FUNCTION_BLOCK EQ_Plunger (* Linear actuator through an L298N (IN1 retract, IN2 extend); no sensors. ENA (200/255 on the ESP32) is tied to 3.3 V on the Pi, which has only two hardware PWM channels, so it runs at full speed; equipment IO: owns its IO points; commands Stop=0, Extend=1, Retract=2 *)
  (* Standard: 61499-2 *)
  (* Version 0.1, 2026-09-28, Project contributors, AAU Smart Production Lab *)
  PACKAGE stoppering;
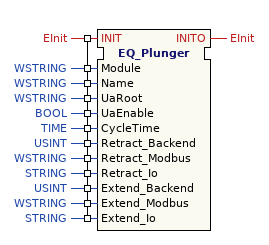
  EVENT_INPUT
    INIT : EInit WITH Module, Name, UaRoot, UaEnable, CycleTime, Retract_Backend, Retract_Modbus, Retract_Io, Extend_Backend, Extend_Modbus, Extend_Io;
  END_EVENT
  EVENT_OUTPUT
    INITO : EInit;
  END_EVENT
  VAR_INPUT
    Module : WSTRING;
    Name : WSTRING := "Plunger";
    UaRoot : WSTRING;
    UaEnable : BOOL;
    CycleTime : TIME := T#50ms;
    Retract_Backend : USINT := 2;
    Retract_Modbus : WSTRING;
    Retract_Io : STRING;
    Extend_Backend : USINT := 2;
    Extend_Modbus : WSTRING;
    Extend_Io : STRING;
  END_VAR
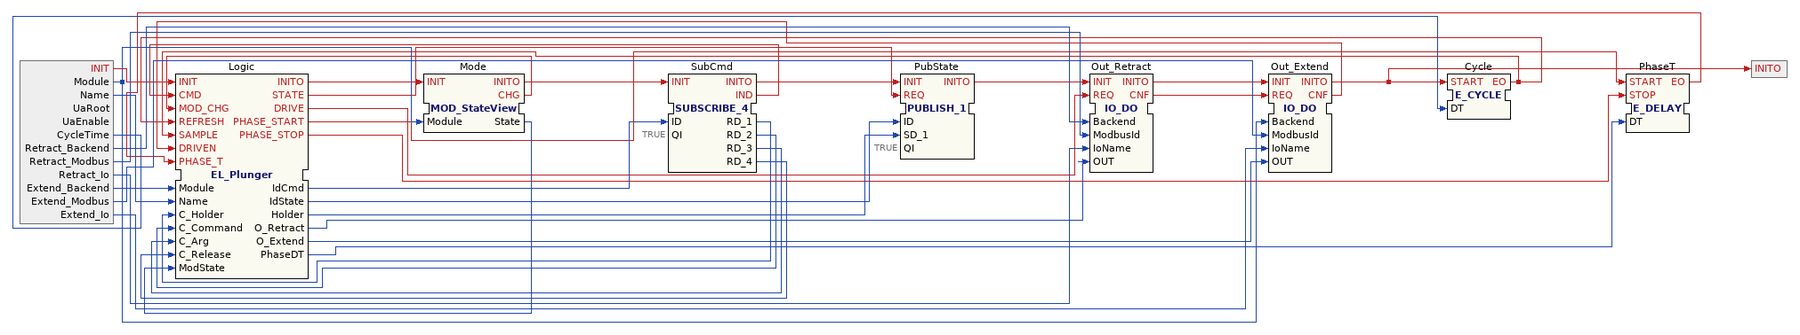
  FBS
    Logic : stoppering::EL_Plunger;
    Mode : modlib::MOD_StateView;
    SubCmd : iec61499::net::SUBSCRIBE_4(QI := TRUE);
    PubState : iec61499::net::PUBLISH_1(QI := TRUE);
    Out_Retract : modlib::IO_DO;
    Out_Extend : modlib::IO_DO;
    Cycle : iec61499::events::E_CYCLE;
    PhaseT : iec61499::events::E_DELAY;
  END_FBS
  EVENT_CONNECTIONS
    INIT TO Logic.INIT;
    Logic.INITO TO Mode.INIT;
    Mode.INITO TO SubCmd.INIT;
    SubCmd.INITO TO PubState.INIT;
    PubState.INITO TO Out_Retract.INIT;
    Out_Retract.INITO TO Out_Extend.INIT;
    Out_Extend.INITO TO Cycle.START;
    Out_Extend.INITO TO INITO;
    SubCmd.IND TO Logic.CMD;
    Mode.CHG TO Logic.MOD_CHG;
    Cycle.EO TO Logic.REFRESH;
    Cycle.EO TO Logic.SAMPLE;
    Logic.STATE TO PubState.REQ;
    Logic.DRIVE TO Out_Retract.REQ;
    Out_Retract.CNF TO Out_Extend.REQ;
    Out_Extend.CNF TO Logic.DRIVEN;
    Logic.PHASE_START TO PhaseT.START;
    Logic.PHASE_STOP TO PhaseT.STOP;
    PhaseT.EO TO Logic.PHASE_T;
  END_CONNECTIONS
  DATA_CONNECTIONS
    Module TO Logic.Module;
    Name TO Logic.Name;
    Module TO Mode.Module;
    Logic.IdCmd TO SubCmd.ID;
    Logic.IdState TO PubState.ID;
    CycleTime TO Cycle.DT;
    SubCmd.RD_1 TO Logic.C_Holder;
    SubCmd.RD_2 TO Logic.C_Command;
    SubCmd.RD_3 TO Logic.C_Arg;
    SubCmd.RD_4 TO Logic.C_Release;
    Mode.State TO Logic.ModState;
    Logic.Holder TO PubState.SD_1;
    Retract_Backend TO Out_Retract.Backend;
    Retract_Modbus TO Out_Retract.ModbusId;
    Retract_Io TO Out_Retract.IoName;
    Logic.O_Retract TO Out_Retract.OUT;
    Extend_Backend TO Out_Extend.Backend;
    Extend_Modbus TO Out_Extend.ModbusId;
    Extend_Io TO Out_Extend.IoName;
    Logic.O_Extend TO Out_Extend.OUT;
    Logic.PhaseDT TO PhaseT.DT;
  END_CONNECTIONS
END_FUNCTION_BLOCK
